FUNCTION_BLOCK FB_Ref_ramp
VAR_INPUT
	Speed_req_in:REAL;
	Allowed_speed:REAL;
	Rate:REAL;
	Zero:BOOL;
	S_Func_scans:REAL;
END_VAR
VAR_OUTPUT
	Speed_ref:INT;
END_VAR
VAR
	Speed_req_real: REAL;
	Speed_step: REAL;
	Speed_ref_real: REAL;
	Speed_up: BOOL;
	FB_CTRL_MOVING_AVERAGE_0: FB_CTRL_MOVING_AVERAGE;
END_VAR
{warning 'TODO: Moving average FB needs to be set up by Bret'}
VAR // added by the converter: edge detectors and wires of the graphical bodies
    _w1, _w3, _w6, _w7 : ANY;
    _w2 : BOOL;
    _w4, _w5, _w8, _w9 : REAL;
END_VAR

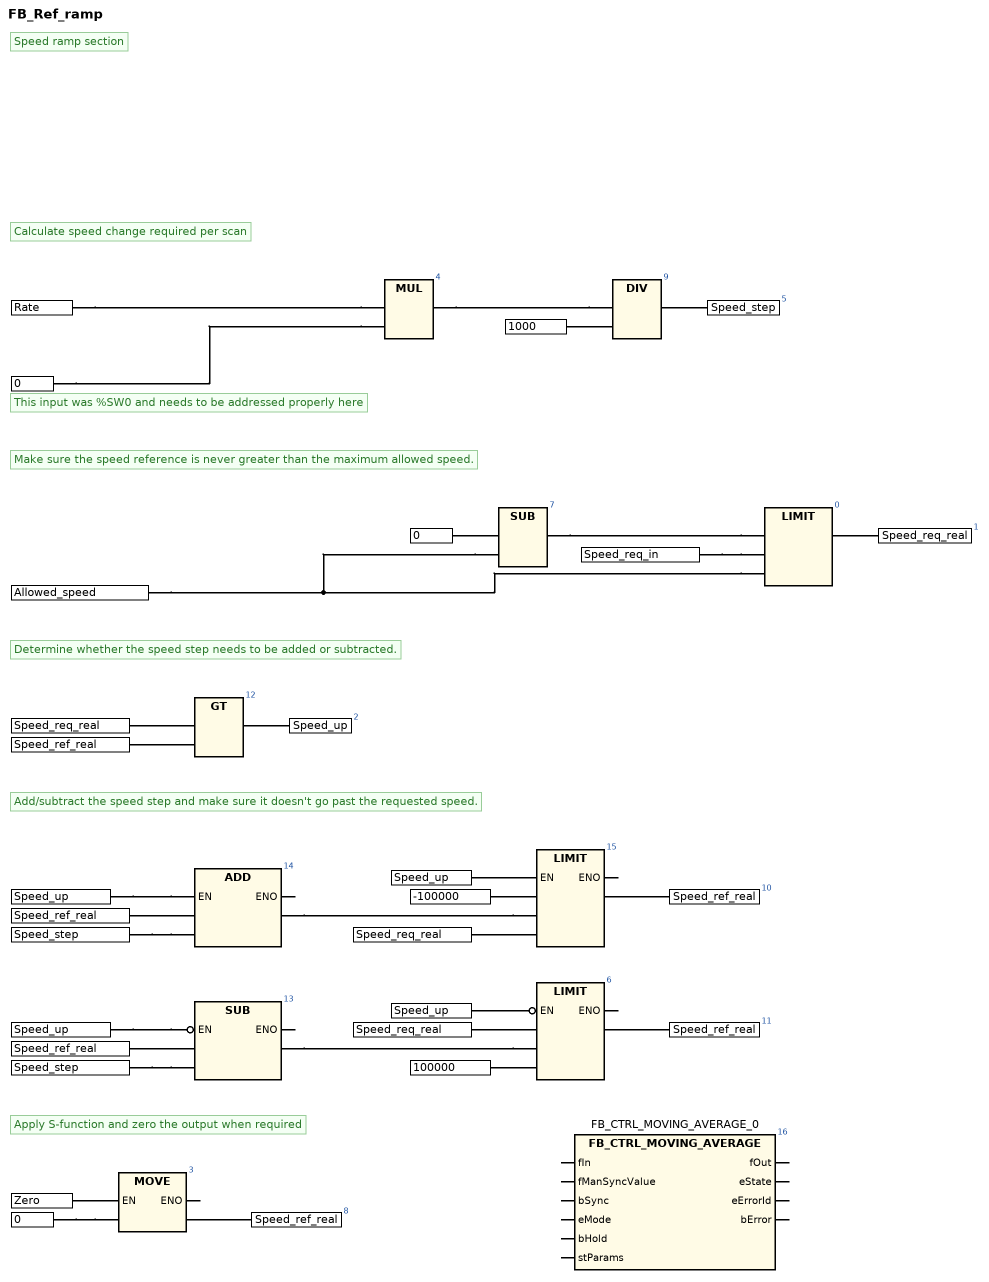
Speed_req_real := LIMIT(_w1, Speed_req_in, Allowed_speed);
Speed_up := _w2;
// Apply S-function and zero the output when required
IF Zero THEN _w3 := 0; END_IF
// Speed ramp section
// Calculate speed change required per scan
_w4 := Rate * 0;
Speed_step := _w5;
IF NOT Speed_up THEN _w7 := LIMIT(Speed_req_real, _w6, 100000); END_IF
// This input was %SW0 and needs to be addressed properly here
// Make sure the speed reference is never greater than the maximum allowed speed.
_w1 := 0 - Allowed_speed;
Speed_ref_real := _w3;
_w5 := _w4 / 1000;
Speed_ref_real := _w8;
Speed_ref_real := _w7;
// Determine whether the speed step needs to be added or subtracted.
_w2 := Speed_req_real > Speed_ref_real;
IF NOT Speed_up THEN _w6 := Speed_ref_real - Speed_step; END_IF
// Add/subtract the speed step and make sure it doesn't go past the requested speed.
IF Speed_up THEN _w9 := Speed_ref_real + Speed_step; END_IF
IF Speed_up THEN _w8 := LIMIT(-100000, _w9, Speed_req_real); END_IF
FB_CTRL_MOVING_AVERAGE_0(); // FB_CTRL_MOVING_AVERAGE

END_FUNCTION_BLOCK

(* stored: Version 1.1.0.1, ProductVersion 3.1.4024.0
   POU FB_Ref_ramp: Id {608e08de-3205-4600-9ab4-8b35700b6efb}, SpecialFunc None *)
